// TIA Portal V18 export
// export: Created 2025-12-01T12:38:01.582756Z, ExportSetting None, DisplayName Totally Integrated Automation Portal, DisplayVersion V18 Update 5, DisplayName TIA Portal Openness, DisplayVersion V18 Update 5, DisplayName TIA Portal Teamcenter Gateway, DisplayVersion V18, DisplayName TIA Portal Version Control Interface, DisplayVersion V18, DisplayName STEP 7 Professional, DisplayVersion V18 Update 5, DisplayName STEP 7 Safety, DisplayVersion V18, DisplayName WinCC Professional, DisplayVersion V18 Update 5
FUNCTION_BLOCK "PartDataManage"   // FB2, SCL
{ S7_Optimized_Access := 'TRUE' }
// stored: MemoryReserve 100, SetENOAutomatically false
   VAR_INPUT
      iReset : Bool;   // 复位
      iScannerTrigger : Bool;   // 扫码枪触发
      iStringRecived : String;   // 扫码枪接收到的物料码
      iMaterialType : String;   // 设定的物料型号
      iSaveToBuffer : Bool;   // 触发将物料信息存储到缓存
      iCodeType : Bool;   // 物料码类型：0，批次码，1，单件码
      iDecrementCnt : DInt := 1;   // 每次的用量
      iDecrementTrigger : Bool;   // 触发信号
      iBufferBoxes : Int := 1;   // 允许缓存的数量,最小为1，最大5
   END_VAR
   VAR_IN_OUT
      ioMaterialActive : Bool;   // 物料比对成功
      io_MaterialManage : "PartData_UDT";
   END_VAR
   VAR
      NO : Array[0..6] of Int;
      sString_MId : String;
      sKeyChar : Char := '#';
      Puls : Array[0..20] of Bool;
      R_TRIG_MaterialActive { S7_SetPoint := 'True'} : R_TRIG;
      R_TRIG_ScannerTrigger { S7_SetPoint := 'True'} : R_TRIG;
      IEC_Timer_MaterialActive { S7_SetPoint := 'True'} : TON_TIME;
      R_TRIG_DecrementTrigger { S7_SetPoint := 'True'} : R_TRIG;
      "R_TRIG_PartQuality+1" { S7_SetPoint := 'True'} : R_TRIG;
      "R_TRIG_PartQuality-1" { S7_SetPoint := 'True'} : R_TRIG;
      R_TRIG_ClearCurrentBox { S7_SetPoint := 'True'} : R_TRIG;
      R_TRIG_ClearAllBox { S7_SetPoint := 'True'} : R_TRIG;
      R_TRIG_SaveToBuffer { S7_SetPoint := 'True'} : R_TRIG;
      Timer_PartQualityAckPB { S7_SetPoint := 'True'} : TON_TIME;
   END_VAR
   VAR_TEMP
      tMaterialTypePos : Int;   // 设定物料码在接收码中的位置
      tLenString : Int;
      BufferIndex : Int;
      "BufferIndex+1" : Int;
      "BufferBoxes-1" : Int;
   END_VAR
BEGIN

   REGION Comment
       //本功能块针对豫北物料编码规则编写，其他项目或规则不宜直接引用：
       //本物料针对手持扫码枪需要扫多个物料的情况，
       //针对物料分为两种：
       //一：单件扫码，物料具有独立标识码，需要将变量  iCodeType  赋 true
       //同时，无需关注其他物料码解析，缓存等功能，
       //只使用    #iStringRecived / #ioMaterialActive 等变量，供程序判断扫码结果和获取物料码使用；
       //不需要配合使用HMI面板
       //二：物料为批次码，需要根据实际情况，设定缓存数量 #iBufferBoxes
       //同时根据需要创建使用HMI面板  
   END_REGION

   REGION 物料比对成功

       #R_TRIG_ScannerTrigger(CLK := #iScannerTrigger);

       #tMaterialTypePos := FIND(IN1 := #iStringRecived, IN2 := #iMaterialType);

       IF #R_TRIG_ScannerTrigger.Q AND #tMaterialTypePos <> 0 THEN
           #ioMaterialActive := 1;
       END_IF;
       //上升沿信号
       #R_TRIG_MaterialActive(CLK := #ioMaterialActive);

       //延时复位
       //
       #IEC_Timer_MaterialActive(IN := #ioMaterialActive,
                                 PT := T#300ms);

       IF #IEC_Timer_MaterialActive.Q THEN
           #ioMaterialActive := 0;
       END_IF;


   END_REGION

   REGION Recive Part Data Analysis

       IF #R_TRIG_MaterialActive.Q AND NOT #iCodeType THEN

           //PartCode
           #io_MaterialManage.PartBoxDataRecive.PartCode := #iStringRecived;
           #io_MaterialManage.PartBoxDataRecive.PartCode_Len := LEN(#io_MaterialManage.PartBoxDataRecive.PartCode);


           //SupplierID
           #NO[0] := FIND(IN1 := #iStringRecived, IN2 := #sKeyChar);
           #NO[1] := #NO[0] - 1;
           #io_MaterialManage.PartBoxDataRecive.SupplierID := LEFT(IN := #iStringRecived, L := #NO[1]);

           //MaterialType
           #tLenString := #io_MaterialManage.PartBoxDataRecive.PartCode_Len - #NO[0];
           #sString_MId := RIGHT_STRING(IN := #iStringRecived, L := #tLenString);
           #NO[0] := FIND(IN1 := #sString_MId, IN2 := #sKeyChar);
           #NO[2] := #NO[0] - 1;
           #io_MaterialManage.PartBoxDataRecive.MaterialType := LEFT(IN := #sString_MId, L := #NO[2]);

           //PO_ID
           //
           #tLenString := #tLenString - #NO[0];
           #sString_MId := RIGHT_STRING(IN := #sString_MId, L := #tLenString);
           #NO[0] := FIND(IN1 := #sString_MId, IN2 := #sKeyChar);
           #NO[3] := #NO[0] - 1;
           #io_MaterialManage.PartBoxDataRecive.PO_ID := LEFT(IN := #sString_MId, L := #NO[3]);

           //BatchID

           #tLenString := #tLenString - #NO[0];
           #sString_MId := RIGHT_STRING(IN := #sString_MId, L := #tLenString);
           #NO[0] := FIND(IN1 := #sString_MId, IN2 := #sKeyChar);
           #NO[4] := #NO[0] - 1;
           #io_MaterialManage.PartBoxDataRecive.BatchID := LEFT(IN := #sString_MId, L := #NO[4]);

           //Quality

           #tLenString := #tLenString - #NO[0];
           #sString_MId := RIGHT_STRING(IN := #sString_MId, L := #tLenString);
           #NO[0] := FIND(IN1 := #sString_MId, IN2 := #sKeyChar);
           #NO[5] := #NO[0] - 1;
           #io_MaterialManage.PartBoxDataRecive.Quality := LEFT(IN := #sString_MId, L := #NO[5]);

           //Cartons
           //
           #tLenString := #tLenString - #NO[0];
           #sString_MId := RIGHT_STRING(IN := #sString_MId, L := #tLenString);
           #io_MaterialManage.PartBoxDataRecive.Cartons := #sString_MId;

       END_IF;
   END_REGION

   REGION Waring
       //物料码已使用，扫码无效   
       IF #ioMaterialActive AND NOT #iCodeType THEN
           IF #io_MaterialManage.PartBoxDataRecive.PartCode = #io_MaterialManage.PartBoxData[1].PartCode
               OR #io_MaterialManage.PartBoxDataRecive.PartCode = #io_MaterialManage.PartBoxData[2].PartCode
               OR #io_MaterialManage.PartBoxDataRecive.PartCode = #io_MaterialManage.PartBoxData[3].PartCode
               OR #io_MaterialManage.PartBoxDataRecive.PartCode = #io_MaterialManage.PartBoxData[4].PartCode
               OR #io_MaterialManage.PartBoxDataRecive.PartCode = #io_MaterialManage.PartBoxData[5].PartCode THEN

               #io_MaterialManage.PartDataHMI.Waring.ScannCodeInvalid := 1;

           END_IF;

       END_IF;


       //物料缓存已满，无法保存
       IF #ioMaterialActive
           AND #io_MaterialManage.PartBoxData[#iBufferBoxes] <> #io_MaterialManage.PartBoxDataNull THEN
           #io_MaterialManage.PartDataHMI.Waring.BufferBoxFull := 1;

       END_IF;
       //物料不足，请及时添加

       IF #io_MaterialManage.PartDataHMI.PartQuality <= #iDecrementCnt THEN
           #io_MaterialManage.PartDataHMI.Waring.Insufficient := 1;

       END_IF;



       IF #iReset THEN

           #io_MaterialManage.PartDataHMI.Waring.Insufficient := 0;
           #io_MaterialManage.PartDataHMI.Waring.BufferBoxFull := 0;
           #io_MaterialManage.PartDataHMI.Waring.ScannCodeInvalid := 0;

       END_IF;

   END_REGION

   REGION Part Data Load LOOP
       IF NOT #iCodeType THEN

           IF #io_MaterialManage.PartDataHMI.PartQuality < #iDecrementCnt THEN

               #io_MaterialManage.PartBoxData[0] := #io_MaterialManage.PartBoxData[1];

               #io_MaterialManage.PartDataHMI.PartQuality := STRING_TO_DINT(IN := #io_MaterialManage.PartBoxData[0].Quality);


               #io_MaterialManage.PartBoxData[1] := #io_MaterialManage.PartBoxDataNull;

           END_IF;


           IF #iBufferBoxes > 1 THEN
               #BufferIndex := 1;
               #"BufferBoxes-1" := #iBufferBoxes - 1;
               FOR #BufferIndex := 1 TO #iBufferBoxes - 1 DO

                   #"BufferIndex+1" := #BufferIndex + 1;

                   IF #io_MaterialManage.PartBoxData[#BufferIndex] = #io_MaterialManage.PartBoxDataNull THEN

                       #io_MaterialManage.PartBoxData[#BufferIndex] := #io_MaterialManage.PartBoxData[#"BufferIndex+1"];

                       #io_MaterialManage.PartBoxData[#"BufferIndex+1"] := #io_MaterialManage.PartBoxDataNull;
                   END_IF;

               END_FOR;

           END_IF;

       END_IF;


       #R_TRIG_SaveToBuffer(CLK:=#iSaveToBuffer);



       IF #R_TRIG_SaveToBuffer.Q AND NOT #iCodeType AND NOT #io_MaterialManage.PartDataHMI.Waring.ScannCodeInvalid
           AND #io_MaterialManage.PartBoxData[#iBufferBoxes] = #io_MaterialManage.PartBoxDataNull THEN

           #io_MaterialManage.PartBoxData[#iBufferBoxes] := #io_MaterialManage.PartBoxDataRecive;

           #io_MaterialManage.PartBoxDataRecive := #io_MaterialManage.PartBoxDataNull;
       END_IF;
   END_REGION

   REGION Part quality 
       //Part quality Decrement
       #R_TRIG_DecrementTrigger(CLK := #iDecrementTrigger);
       IF #R_TRIG_DecrementTrigger.Q THEN
           #io_MaterialManage.PartDataHMI.PartQuality := #io_MaterialManage.PartDataHMI.PartQuality - #iDecrementCnt;
       END_IF;

      // Part quality Adjust
       #"R_TRIG_PartQuality+1"(CLK:=#io_MaterialManage.PartDataHMI.CMD."PartQuality+1");
       #"R_TRIG_PartQuality-1"(CLK:=#io_MaterialManage.PartDataHMI.CMD."PartQuality-1");

       IF #"R_TRIG_PartQuality+1".Q THEN
           #io_MaterialManage.PartDataHMI.PartQuality :=#io_MaterialManage.PartDataHMI.PartQuality + 1;
       END_IF;
       IF #"R_TRIG_PartQuality-1".Q THEN
           #io_MaterialManage.PartDataHMI.PartQuality := #io_MaterialManage.PartDataHMI.PartQuality - 1;

       END_IF;

       // Part quality Set By Operator
       #Timer_PartQualityAckPB(IN:=#io_MaterialManage.PartDataHMI.CMD.PartQualityAck,
                               PT:=t#2s);

       IF #Timer_PartQualityAckPB.Q THEN

           #io_MaterialManage.PartDataHMI.PartQuality := #io_MaterialManage.PartDataHMI.PartQualitySet;
       END_IF;




       // Part Data Clear
       #R_TRIG_ClearCurrentBox(CLK := #io_MaterialManage.PartDataHMI.CMD.ClearCurrentBox);
       #R_TRIG_ClearAllBox(CLK := #io_MaterialManage.PartDataHMI.CMD.ClearAllBox);

       IF #R_TRIG_ClearCurrentBox.Q THEN
           #io_MaterialManage.PartBoxData[0] := #io_MaterialManage.PartBoxDataNull;

       END_IF;

       IF #R_TRIG_ClearAllBox.Q THEN

           #BufferIndex := 0;
           FOR #BufferIndex := 0 TO 20 DO
               #io_MaterialManage.PartBoxData[#BufferIndex] := #io_MaterialManage.PartBoxDataNull;
           END_FOR;
       END_IF;

   END_REGION


   REGION PartData Dispaly
       #io_MaterialManage.PartDataHMI.PartDataDispaly := #io_MaterialManage.PartBoxData[#io_MaterialManage.PartDataHMI.BoxDisplayID];
   END_REGION
END_FUNCTION_BLOCK
